FUNCTION_BLOCK IntegralController
  (* Standard: 61499-2 *)
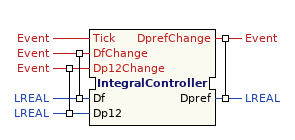
  EVENT_INPUT
    Tick;
    DfChange WITH Df;
    Dp12Change WITH Dp12;
  END_EVENT
  EVENT_OUTPUT
    DprefChange WITH Dpref;
  END_EVENT
  VAR_INPUT
    Df : LREAL;
    Dp12 : LREAL;
  END_VAR
  VAR_OUTPUT
    Dpref : LREAL;
  END_VAR
  VAR
    StepSize : LREAL := 0.1;
    Ki : LREAL := 0.5;
    B : LREAL := 0.425;
  END_VAR
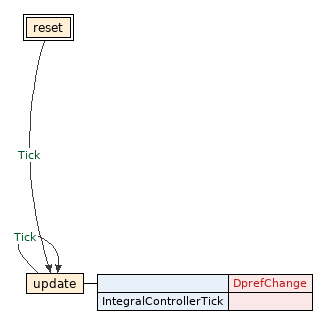
  EC_STATES
    reset;
    update : -> DprefChange, IntegralControllerTick;
  END_STATES
  EC_TRANSITIONS
    reset TO update := Tick;
    update TO update := Tick;
  END_TRANSITIONS
  ALGORITHM IntegralControllerTick IN ST:
        Dpref := Dpref - (Ki * (Df*B + Dp12))*StepSize;
  END_ALGORITHM
END_FUNCTION_BLOCK
